INTERFACE I_TcpIpSubscription EXTENDS I_Base

METHOD UpdateCommandResult
VAR_INPUT
	Response : POINTER TO ST_TcpIpPayload;
END_VAR
END_METHOD

END_INTERFACE

(* stored: Version 1.1.0.1, ProductVersion 3.1.4026.18
   Itf I_TcpIpSubscription: Id {79364947-c7cb-43c7-b2b2-46dcb49b7b8a}
   Method UpdateCommandResult: Id {495997fc-7ab0-481a-9ebe-7ee90f3042a1} *)
